// TIA Portal V17 export
// export: Created 2024-09-02T12:50:41.3477727Z, ExportSetting WithDefaults, DisplayName Totally Integrated Automation Portal, DisplayVersion V17, DisplayName TIA Portal Openness, DisplayVersion V17, DisplayName TIA Portal Version Control Interface, DisplayVersion V17, DisplayName STEP 7 Professional, DisplayVersion V17, DisplayName STEP 7 Safety, DisplayVersion V17, DisplayName WinCC Professional, DisplayVersion V17
TYPE "Aveva_Desutter_Result"
// stored: IsFailsafeCompliant false
   STRUCT
      Status { ExternalWritable := 'False'} : Array[0..7] of Bool;   // %X0-Work Finished NOK/%X1 Work Finished OK /%X2 Work Bypassed /%X3 Work Interrupted
      RetryPreformed { ExternalWritable := 'False'} : Int;   // Number of retry
      Torque { ExternalWritable := 'False'} : Real;   // Value of torque (Nm)
      Angle { ExternalWritable := 'False'} : Real;   // Value of angle (Degree)
   END_STRUCT;
END_TYPE
